// TIA Portal V18 export
DATA_BLOCK "DB_FB_Coveyor_5"   // DB10
VERSION : 0.1
// stored: AutoNumber true, DBAccessibleFromOPCUA true, DBAccessibleFromWebserver true, InstanceOfName FB_Coveyor, InstanceOfType FB
"FB_Coveyor"
   // VAR_INPUT
   //    in_sensor_in : Bool;
   //    in_sensor_out : Bool;
   // END_VAR
   // VAR_OUTPUT
   //    out_busy : Bool;
   // END_VAR
   // VAR
   //    busy : Bool;
   //    cont : Int;
   //    speed : Int;
   // END_VAR
BEGIN
END_DATA_BLOCK
